// TIA Portal project "Hardware" (V14)

(* hardware
DEVICE "ET 200S-Station_1"  ET 200S station
   slot 0: "Baugruppenträger_0"  Rail
   slot 2: "PLC_1"  IM151-8 CPU  6ES7 151-8AB00-0AB0  V2.7
      slot 1: "PROFINET-Schnittstelle_1"  PN-IO
         slot 1: "Port_1"  Port
         slot 2: "Port_2"  Port
         slot 3: "Port_3"  Port
   slot 4: "PM-E 24VDC_1"  PM-E 24VDC  6ES7 138-4CA01-0AA0
   slot 5: "4AI x I 2WIRE ST_1"  4AI x I 2WIRE ST  6ES7 134-4GD00-0AB0
   slot 6: "2AO x U ST_1"  2AO x U ST  6ES7 135-4FB01-0AB0
   slot 7: "8DI x 24VDC_1"  8DI x 24VDC  6ES7 131-4BF00-0AA0
   slot 8: "8DI x 24VDC_2"  8DI x 24VDC  6ES7 131-4BF00-0AA0
   slot 9: "8DI x 24VDC_3"  8DI x 24VDC  6ES7 131-4BF00-0AA0
   slot 10: "8DI x 24VDC_4"  8DI x 24VDC  6ES7 131-4BF00-0AA0
   slot 11: "8DO x 24VDC / 0.5A_1"  8DO x 24VDC / 0.5A  6ES7 132-4BF00-0AA0
   slot 12: "8DO x 24VDC / 0.5A_2"  8DO x 24VDC / 0.5A  6ES7 132-4BF00-0AA0
   slot 13: "8DO x 24VDC / 0.5A_3"  8DO x 24VDC / 0.5A  6ES7 132-4BF00-0AA0
   slot 14: "8DO x 24VDC / 0.5A_4"  8DO x 24VDC / 0.5A  6ES7 132-4BF00-0AA0
DEVICE "HMI_1"  TP 177B 6'' PN/DP
   slot 0: "TP 177B 6'' PN/DP"  TP 177B 6'' PN/DP  6AV6 642-0BA01-1AX1  11.0.2.0
   slot 1: "HMI_RT_1"  TP 177B 6'' PN/DP  6AV6 642-0BA01-1AX1  11.0.2.0
   slot 5: "HMI_1.IE_CP_1"  PROFINET Interface  11.0.0.0
      slot 1: "PROFINET Schnittstelle_1"  PROFINET Interface
         slot 1: "Port_1"  Port
   slot 7: "HMI_1.MPI/DP_CP_1"  MPI/DP Interface  11.0.0.0
*)

// ===== PLC "PLC_1"  IM151-8 CPU =====

VAR_GLOBAL   // PLC tag table "Standard-Variablentabelle"
   "Blinken" AT %A7.0 : Bool;
   "Sekundentakt" AT %M100.5 : Bool;
   "A_rot" AT %A9.6 : Bool;
   "A_gelb" AT %A9.7 : Bool;
   "A_gruen" AT %A10.0 : Bool;
   "F_rot" AT %A10.6 : Bool;
   "F_gruen" AT %A10.7 : Bool;
   "Tag_1" AT %M0.0 : Bool;
   "Zweisekundentakt" AT %M100.7 : Bool;
   "Tag_2" AT %M3.0 : Bool;
   "Tag_3" AT %MD12 : DWord;
   "Tag_4" AT %MD16 : DWord;
   "Tag_5" AT %MW20 : Int;
   "Tag_6" AT %MW21 : Int;
   "Tag_7" AT %MW30 : Int;
   "Tag_8" AT %M22.7 : Bool;
   "Tag_9" AT %M2.0 : Bool;
END_VAR

DATA_BLOCK "Tagbetrieb_fb_DB"   // DB2
{ S7_Optimized_Access := 'FALSE' }
VERSION : 0.1
// stored: InstanceOfName Tagbetrieb_fb
"Tagbetrieb_fb"
BEGIN
END_DATA_BLOCK

DATA_BLOCK "Variable"   // DB3
{ S7_Optimized_Access := 'FALSE' }
VERSION : 0.1
   VAR
      Tag : Bool;
      Zeit : Int;
   END_VAR
BEGIN
END_DATA_BLOCK

FUNCTION_BLOCK "Tagbetrieb_fb"   // FB1, FBD
{ S7_Optimized_Access := 'FALSE' }
VERSION : 0.1
   VAR_INPUT
      Sekundentakt : Bool;
   END_VAR
   VAR_OUTPUT
      Auto_rot : Bool;
      Auto_gelb : Bool;
      Auto_gruen : Bool;
      FG_rot : Bool;
      FG_gruen : Bool;
   END_VAR
   VAR
      S5 : Bool;
   END_VAR
   VAR_TEMP
      S1 : Bool;
      S2 : Bool;
      S3 : Bool;
      S4 : Bool;
      Zaehler : Int;
   END_VAR
BEGIN

REGION Network 1
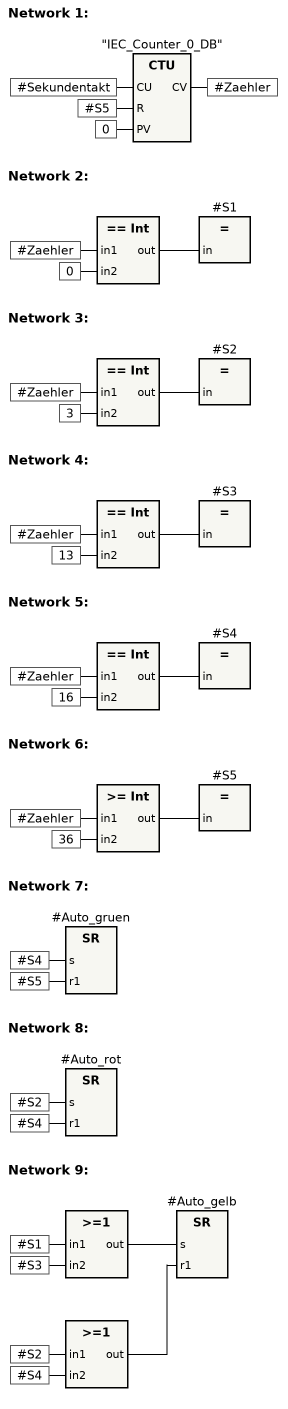
   "IEC_Counter_0_DB".CTU(CU := #Sekundentakt, R := #S5, PV := 0, CV => #Zaehler);
END_REGION

REGION Network 2
   #S1 := #Zaehler = 0;
END_REGION

REGION Network 3
   #S2 := #Zaehler = 3;
END_REGION

REGION Network 4
   #S3 := #Zaehler = 13;
END_REGION

REGION Network 5
   #S4 := #Zaehler = 16;
END_REGION

REGION Network 6
   #S5 := #Zaehler >= 36;
END_REGION

REGION Network 7
   IF #S4 THEN
       #Auto_gruen := TRUE;   // SR flip-flop
   END_IF;
   IF #S5 THEN #Auto_gruen := FALSE; END_IF;
END_REGION

REGION Network 8
   IF #S2 THEN
       #Auto_rot := TRUE;   // SR flip-flop
   END_IF;
   IF #S4 THEN #Auto_rot := FALSE; END_IF;
END_REGION

REGION Network 9
   IF #S1 OR #S3 THEN
       #Auto_gelb := TRUE;   // SR flip-flop
   END_IF;
   IF #S2 OR #S4 THEN #Auto_gelb := FALSE; END_IF;
END_REGION

REGION Network 10
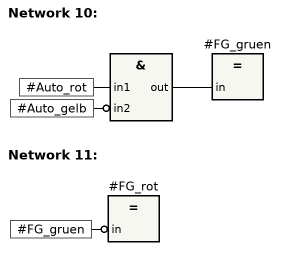
   #FG_gruen := #Auto_rot AND NOT #Auto_gelb;
END_REGION

REGION Network 11
   #FG_rot := NOT #FG_gruen;
END_REGION
END_FUNCTION_BLOCK

FUNCTION "Tagbetrieb" : Void   // FC1, FBD
{ S7_Optimized_Access := 'FALSE' }
VERSION : 0.1
   VAR_INPUT
      Sekundentakt : Bool;
   END_VAR
   VAR_OUTPUT
      Auto_rot : Bool;
      Auto_gelb : Bool;
      Auto_gruen : Bool;
      FG_rot : Bool;
      FG_gruen : Bool;
   END_VAR
   VAR_TEMP
      S1 : Bool;
      S2 : Bool;
      S3 : Bool;
      S4 : Bool;
      S5 : Bool;
      Zaehler : Int;
   END_VAR
BEGIN

REGION Network 1
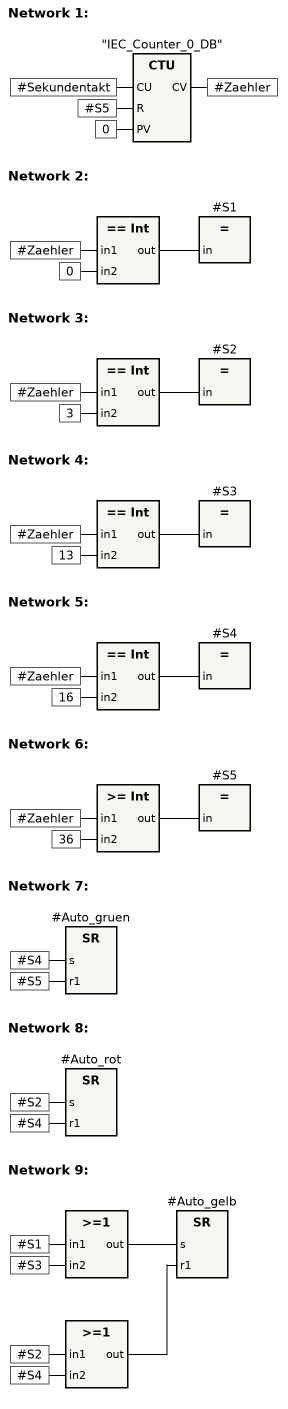
   "IEC_Counter_0_DB".CTU(CU := #Sekundentakt, R := #S5, PV := 0, CV => #Zaehler);
END_REGION

REGION Network 2
   #S1 := #Zaehler = 0;
END_REGION

REGION Network 3
   #S2 := #Zaehler = 3;
END_REGION

REGION Network 4
   #S3 := #Zaehler = 13;
END_REGION

REGION Network 5
   #S4 := #Zaehler = 16;
END_REGION

REGION Network 6
   #S5 := #Zaehler >= 36;
END_REGION

REGION Network 7
   IF #S4 THEN
       #Auto_gruen := TRUE;   // SR flip-flop
   END_IF;
   IF #S5 THEN #Auto_gruen := FALSE; END_IF;
END_REGION

REGION Network 8
   IF #S2 THEN
       #Auto_rot := TRUE;   // SR flip-flop
   END_IF;
   IF #S4 THEN #Auto_rot := FALSE; END_IF;
END_REGION

REGION Network 9
   IF #S1 OR #S3 THEN
       #Auto_gelb := TRUE;   // SR flip-flop
   END_IF;
   IF #S2 OR #S4 THEN #Auto_gelb := FALSE; END_IF;
END_REGION

REGION Network 10
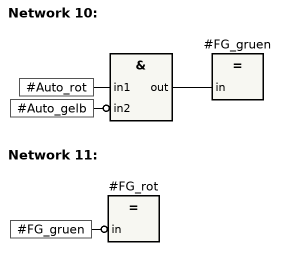
   #FG_gruen := #Auto_rot AND NOT #Auto_gelb;
END_REGION

REGION Network 11
   #FG_rot := NOT #FG_gruen;
END_REGION
END_FUNCTION

FUNCTION "Nachtbetrieb" : Void   // FC2, FBD
{ S7_Optimized_Access := 'FALSE' }
VERSION : 0.1
   VAR_INPUT
      Zweisekundentakt : Bool;
   END_VAR
   VAR_OUTPUT
      Auto_rot : Bool;
      Auto_gelb : Bool;
      Auto_gruen : Bool;
      FG_rot : Bool;
      FG_gruen : Bool;
   END_VAR
BEGIN

REGION Network 1
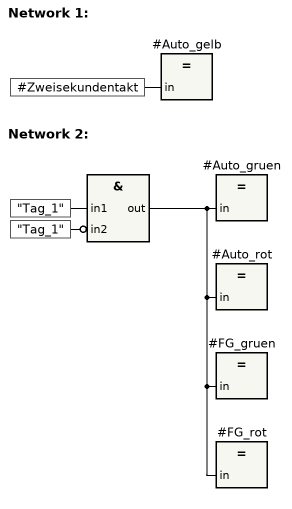
   #Auto_gelb := #Zweisekundentakt;
END_REGION

REGION Network 2
   #Auto_gruen := "Tag_1" AND NOT "Tag_1";
   #Auto_rot := #Auto_gruen;
   #FG_gruen := #Auto_gruen;
   #FG_rot := #Auto_gruen;
END_REGION
END_FUNCTION

FUNCTION "Minuten_des_Tages" : Int   // FC3, FBD
{ S7_Optimized_Access := 'FALSE' }
VERSION : 0.1
   VAR_INPUT
      Std : Byte;
      Min : Byte;
   END_VAR
   VAR_TEMP
      Std_w : Word;
      Std_i : Int;
      Min_w : Word;
      Min_i : Int;
      std_mal_60 : Int;
   END_VAR
BEGIN

REGION Network 1
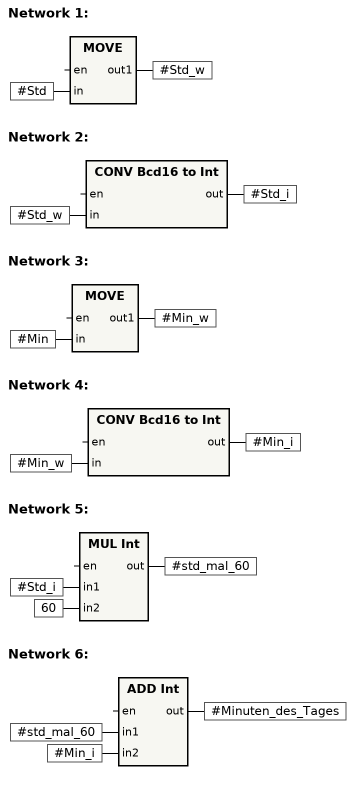
   #Std_w := #Std;
END_REGION

REGION Network 2
   #Std_i := BCD16_TO_INT(#Std_w);
END_REGION

REGION Network 3
   #Min_w := #Min;
END_REGION

REGION Network 4
   #Min_i := BCD16_TO_INT(#Min_w);
END_REGION

REGION Network 5
   #std_mal_60 := #Std_i * 60;
END_REGION

REGION Network 6
   #Minuten_des_Tages := #std_mal_60 + #Min_i;
END_REGION
END_FUNCTION

ORGANIZATION_BLOCK "Main"   // OB1, FBD
TITLE = "Main Program Sweep (Cycle)"
{ S7_Optimized_Access := 'FALSE' }
VERSION : 0.1
   VAR_TEMP
      OB1_EV_CLASS : Byte;   // Bits 0-3 = 1 (Coming event), Bits 4-7 = 1 (Event class 1)
      OB1_SCAN_1 : Byte;   // 1 (Cold restart scan 1 of OB 1), 3 (Scan 2-n of OB 1)
      OB1_PRIORITY : Byte;   // Priority of OB Execution
      OB1_OB_NUMBR : Byte;   // 1 (Organization block 1, OB1)
      OB1_RESERVED_1 : Byte;   // Reserved for system
      OB1_RESERVED_2 : Byte;   // Reserved for system
      OB1_PREV_CYCLE : Int;   // Cycle time of previous OB1 scan (milliseconds)
      OB1_MIN_CYCLE : Int;   // Minimum cycle time of OB1 (milliseconds)
      OB1_MAX_CYCLE : Int;   // Maximum cycle time of OB1 (milliseconds)
      OB1_DATE_TIME : Date_And_Time;   // Date and time OB1 started
   END_VAR
BEGIN

REGION Network 1
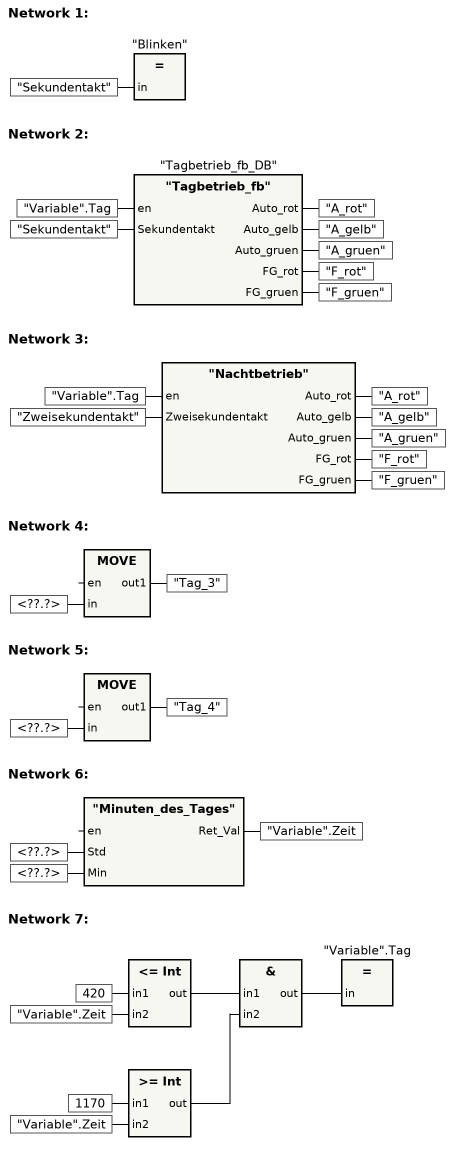
   "Blinken" := "Sekundentakt";
END_REGION

REGION Network 2
   IF "Variable".Tag THEN
       "Tagbetrieb_fb_DB"(Sekundentakt := "Sekundentakt",   // "Tagbetrieb_fb"
                          Auto_rot => "A_rot",
                          Auto_gelb => "A_gelb",
                          Auto_gruen => "A_gruen",
                          FG_rot => "F_rot",
                          FG_gruen => "F_gruen");
   END_IF;
END_REGION

REGION Network 3
   IF "Variable".Tag THEN
       "Nachtbetrieb"(Zweisekundentakt := "Zweisekundentakt",
                      Auto_rot => "A_rot",
                      Auto_gelb => "A_gelb",
                      Auto_gruen => "A_gruen",
                      FG_rot => "F_rot",
                      FG_gruen => "F_gruen");
   END_IF;
END_REGION

REGION Network 4
   "Tag_3" := <??.?>;
END_REGION

REGION Network 5
   "Tag_4" := <??.?>;
END_REGION

REGION Network 6
   "Variable".Zeit := "Minuten_des_Tages"(Std := <??.?>, Min := <??.?>);
END_REGION

REGION Network 7
   "Variable".Tag := (420 <= "Variable".Zeit) AND (1170 >= "Variable".Zeit);
END_REGION
END_ORGANIZATION_BLOCK

(* ===== HMI "HMI_RT_1" =====
system functions are stored by id; their names below are inferred from use
connection "HMI_Verbindung_1": ETHERNET, SIMATIC S7 300/400 MPI
connection "HMI_Verbindung_2": ETHERNET, SIMATIC S7 300/400 MPI

HMI tags "Standard-Variablentabelle"
   "Variable_Bildnummer" : UInt, internal
   "A_rot" : Bool = PLC A_rot AT %A9.6, 1 s
   "A_gelb" : Bool = PLC A_gelb AT %A9.7, 1 s
   "A_gruen" : Bool = PLC A_gruen AT %A10.0, 1 s

text list "Textliste_Bildnamen": 1 'Grundbild'; 2 'Ampel'; 3 'Uhrzeit'

screen "Uhrzeit" 320x200, template "Vorlage_1"
   on GenerateScreen: SetTag("Variable_Bildnummer", 3)
   TextField "HmiScreenItemData" at 32,63 size 256x20; Text 'Uhrzeit'
   Button "Zurück" at 1,1 size 104x36; TextOff 'Zurück'
      on Release: ActivateScreen("Grundbild", 0)

screen "Grundbild" 320x200, template "Vorlage_1"
   on GenerateScreen: SetTag("Variable_Bildnummer", 1)
   TextField "HmiScreenItemData" at 32,55 size 256x36; Text 'Willkommen zum HMI_1 (TP 177B 6″ PN/DP)!'
   Button "Ampel" at 1,1 size 104x36; TextOff 'Ampel'
      on Release: ActivateScreen("Ampel", 0)
   Button "Uhrzeit" at 106,1 size 104x36; TextOff 'Uhrzeit'
      on Release: ActivateScreen("Uhrzeit", 0)

Template "Vorlage_1" 320x200
   Button "Beenden" at 267,150 size 51x47; TextOff 'Beenden'; PictureOff "ExitRuntime_TP_177B_6_PNDP"; PictureOn "ExitRuntime_TP_177B_6_PNDP"
      on Release: StopRuntime(0)
   Button "Template_Button" at 214,150 size 51x47; TextOff 'Text'
   Button "Template_Button_1" at 160,150 size 51x47; TextOff 'Text'
   Button "Template_Button_2" at 107,150 size 51x47; TextOff 'Text'
   Button "Template_Button_3" at 54,150 size 51x47; TextOff 'Text'
   Button "Startbild" at 1,150 size 51x47; TextOff 'Startbild'; PictureOff "NavigateHome_TP_177B_6_PNDP"; PictureOn "NavigateHome_TP_177B_6_PNDP"
      on Release: ActivateScreen("Grundbild", 0)

screen "Ampel" 320x200, template "Vorlage_1"
   on GenerateScreen: SetTag("Variable_Bildnummer", 2)
   GraphicView "Grafikanzeige_1" at 0,1 size 319x148; Picture "strasse"
   Circle "Kreis_1" at 173,7 size 18x18
      Visibility <- "A_rot"
   Circle "Kreis_2" at 192,7 size 18x18
      Appearance <- "A_gelb"
   Circle "Kreis_3" at 211,8 size 18x18
      Visibility <- "A_gruen"
*)